// SIMATIC S7-200 SMART project (STEP 7-Micro/WIN SMART), CPU SR60

SYMBOL_TABLE Table 1
Start_0          M0.1     // Rotate the belt to fill material from the start of the belt
Start_End        M0.2     // Rotate the belt to fill material from the end of the belt
Case1            M0.3
Rotate_F         M1.3     // Rotate the shuttle trolly forward
Case3            M0.5
Case4            M0.6
Case2            M0.4
O1               M1.0
O2               M1.1
SCALED_ANALOG_INPUT VD40
Distance_in_cm   VW10     // Distance calculated by the sensor in centimeters
N1               VW20     // distance between the first sensors and the starting point of the conveyor belt
N2               VW22     // distance between the second sensors and the starting point of the conveyor belt
SENSOR_1         VW100
SENSOR_2         VW102
Rot_CW           M3.0     // Rotate the belt to fill from the start of the belt
Rot_ACW          M3.1     // Rotate the belt to fill from the end of the belt
Rotate_B         M0.7     // Rotate the shuttle trolly backword
END_SYMBOL_TABLE

SYMBOL_TABLE System Symbols
Always_On        SM0.0    // Always ON
END_SYMBOL_TABLE

ORGANIZATION_BLOCK MAIN:OB1
TITLE=Program Comments
BEGIN
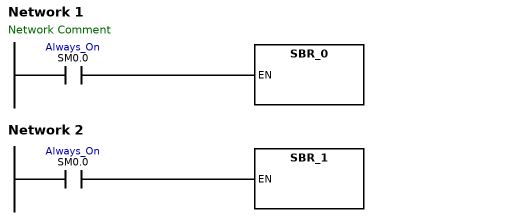
Network 1
// Network Comment
LD     Always_On:SM0.0
CALL   SBR_0:SBR0
Network 2
LD     Always_On:SM0.0
CALL   SBR_1:SBR1
END_ORGANIZATION_BLOCK

SUBROUTINE_BLOCK SBR_0:SBR0
TITLE=Subroutine Comments
BEGIN
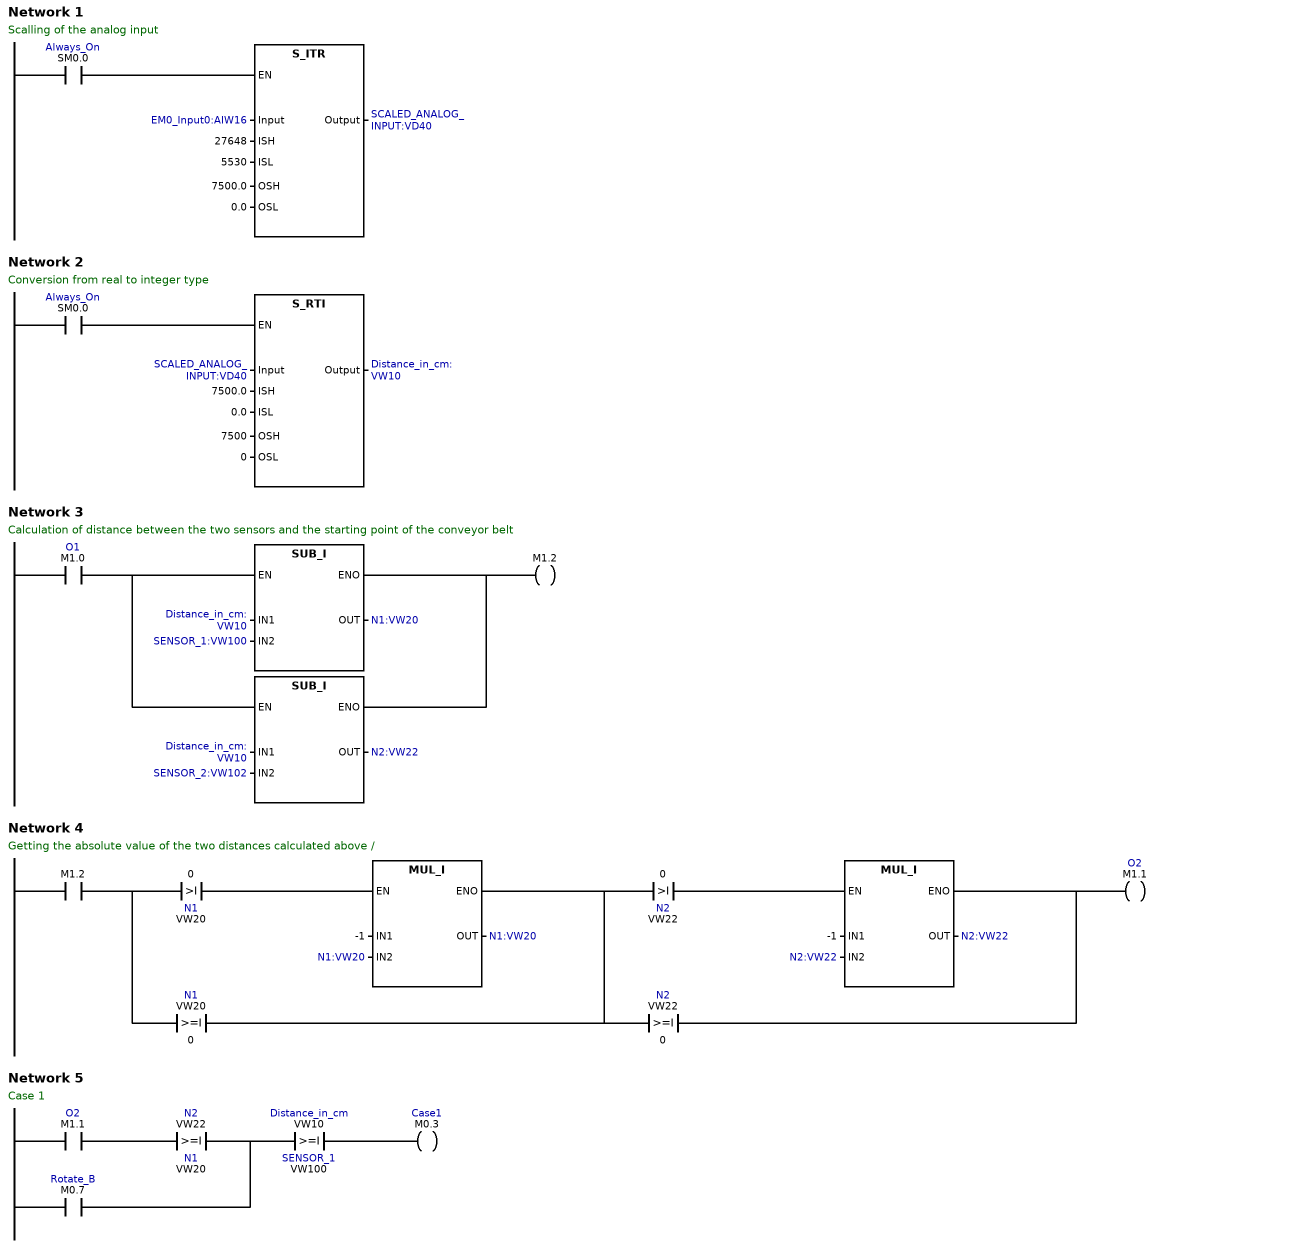
Network 1
// Scalling of the analog input
// (network saved uncompiled; LAD cells follow)
// row 0: c0 -| |- Always_On:SM0.0  c1 --  c2 [S_ITR EN:=power@row0, Input:=EM0_Input0:AIW16, ISH:=27648, ISL:=5530, OSH:=7500.0, OSL:=0.0, Output=>SCALED_ANALOG_INPUT:VD40]
// row 1: c2 [box]
// row 2: c2 [box]
Network 2
// Conversion from real to integer type
// (network saved uncompiled; LAD cells follow)
// row 0: c0 -| |- Always_On:SM0.0  c1 --  c2 [S_RTI EN:=power@row0, Input:=SCALED_ANALOG_INPUT:VD40, ISH:=7500.0, ISL:=0.0, OSH:=7500, OSL:=0, Output=>Distance_in_cm:VW10]
// row 1: c2 [box]
// row 2: c2 [box]
Network 3
// Calculation of distance between the two sensors and the starting point of the conveyor belt
// (network saved uncompiled; LAD cells follow)
// row 0: c0 -| |- O1:M1.0 v  c1 --  c2 [SUB_I EN:=power@row0, IN1:=Distance_in_cm:VW10, IN2:=SENSOR_1:VW100, ENO=>power, OUT=>N1:VW20]  c3 -- v  c4 -( ) M1.2
// row 1: c0 ^v  c2 [box]  c3 ^v
// row 2: c0 ^  c1 --  c2 [SUB_I EN:=power@row2, IN1:=Distance_in_cm:VW10, IN2:=SENSOR_2:VW102, ENO=>power, OUT=>N2:VW22]  c3 -- ^
// row 3: c2 [box]
Network 4
// Getting the absolute value of the two distances calculated above
// 
LD     M1.2
LPS
AW>    0, N1:VW20
*I     -1, N1:VW20
AENO
=      L63.7
LPP
AW>=   N1:VW20, 0
O      L63.7
LPS
AW>    0, N2:VW22
*I     -1, N2:VW22
AENO
=      L63.6
LPP
AW>=   N2:VW22, 0
O      L63.6
=      O2:M1.1
Network 5
// Case 1
// (network saved uncompiled; LAD cells follow)
// row 0: c0 -| |- O2:M1.1  c1 -|>=I|- N2:VW22, N1:VW20 v  c2 -|>=I|- Distance_in_cm:VW10, SENSOR_1:VW100  c3 -( ) Case1:M0.3
// row 1: c0 -| |- Rotate_B:M0.7  c1 -- ^
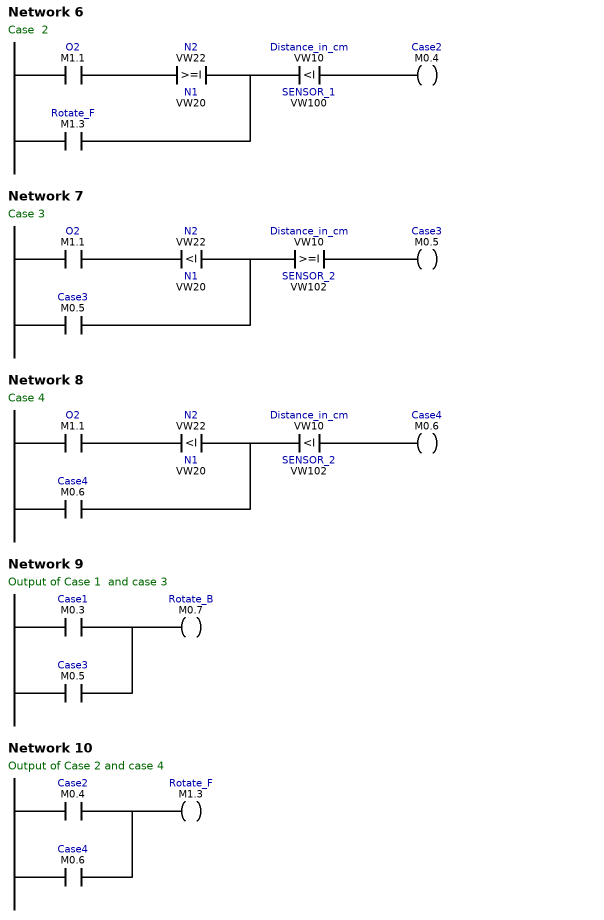
Network 6
// Case  2
// (network saved uncompiled; LAD cells follow)
// row 0: c0 -| |- O2:M1.1  c1 -|>=I|- N2:VW22, N1:VW20 v  c2 -|<I|- Distance_in_cm:VW10, SENSOR_1:VW100  c3 -( ) Case2:M0.4
// row 1: c0 -| |- Rotate_F:M1.3  c1 -- ^
Network 7
// Case 3
// (network saved uncompiled; LAD cells follow)
// row 0: c0 -| |- O2:M1.1  c1 -|<I|- N2:VW22, N1:VW20 v  c2 -|>=I|- Distance_in_cm:VW10, SENSOR_2:VW102  c3 -( ) Case3:M0.5
// row 1: c0 -| |- Case3:M0.5  c1 -- ^
Network 8
// Case 4
// (network saved uncompiled; LAD cells follow)
// row 0: c0 -| |- O2:M1.1  c1 -|<I|- N2:VW22, N1:VW20 v  c2 -|<I|- Distance_in_cm:VW10, SENSOR_2:VW102  c3 -( ) Case4:M0.6
// row 1: c0 -| |- Case4:M0.6  c1 -- ^
Network 9
// Output of Case 1  and case 3
LD     Case1:M0.3
O      Case3:M0.5
=      Rotate_B:M0.7
Network 10
// Output of Case 2 and case 4
LD     Case2:M0.4
O      Case4:M0.6
=      Rotate_F:M1.3
END_SUBROUTINE_BLOCK

SUBROUTINE_BLOCK SBR_1:SBR1
TITLE=Storage and selection of the bunker number
BEGIN
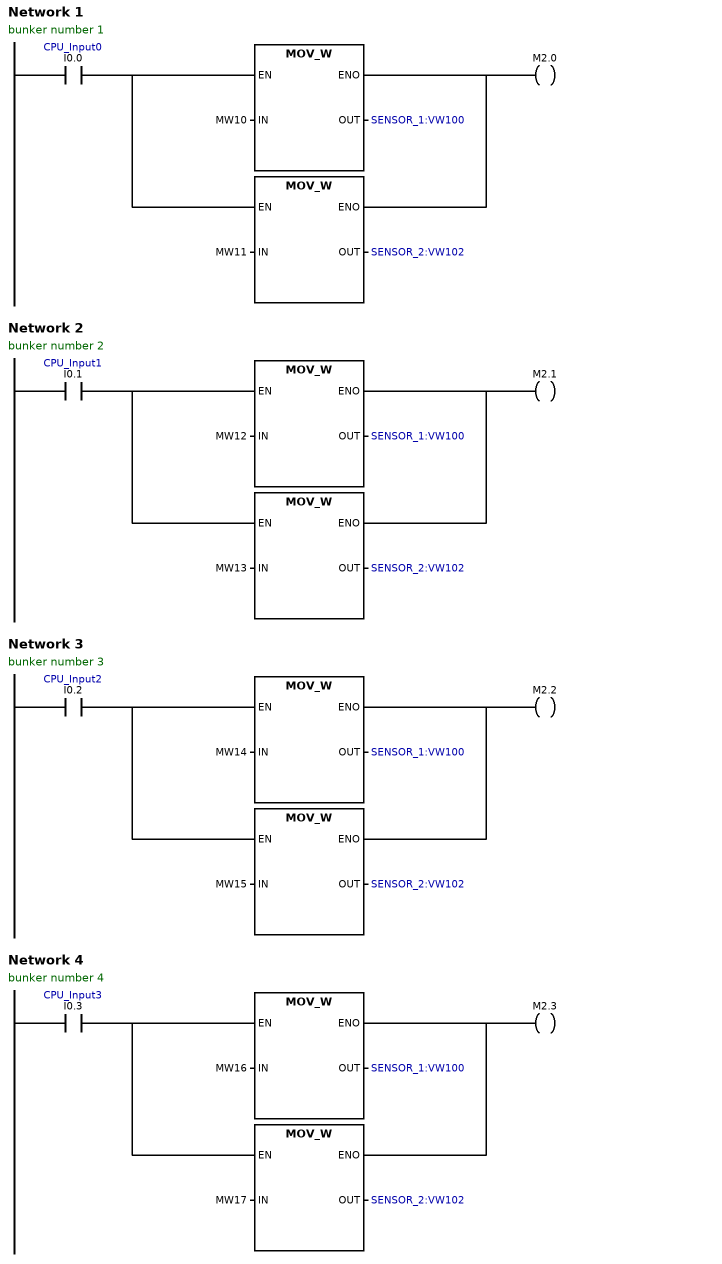
Network 1
// bunker number 1
// (network saved uncompiled; LAD cells follow)
// row 0: c0 -| |- CPU_Input0:I0.0 v  c1 --  c2 [MOV_W EN:=power@row0, IN:=MW10, ENO=>power, OUT=>SENSOR_1:VW100]  c3 -- v  c4 -( ) M2.0
// row 1: c0 ^v  c2 [box]  c3 ^v
// row 2: c0 ^  c1 --  c2 [MOV_W EN:=power@row2, IN:=MW11, ENO=>power, OUT=>SENSOR_2:VW102]  c3 -- ^
// row 3: c2 [box]
Network 2
// bunker number 2
// (network saved uncompiled; LAD cells follow)
// row 0: c0 -| |- CPU_Input1:I0.1 v  c1 --  c2 [MOV_W EN:=power@row0, IN:=MW12, ENO=>power, OUT=>SENSOR_1:VW100]  c3 -- v  c4 -( ) M2.1
// row 1: c0 ^v  c2 [box]  c3 ^v
// row 2: c0 ^  c1 --  c2 [MOV_W EN:=power@row2, IN:=MW13, ENO=>power, OUT=>SENSOR_2:VW102]  c3 -- ^
// row 3: c2 [box]
Network 3
// bunker number 3
// (network saved uncompiled; LAD cells follow)
// row 0: c0 -| |- CPU_Input2:I0.2 v  c1 --  c2 [MOV_W EN:=power@row0, IN:=MW14, ENO=>power, OUT=>SENSOR_1:VW100]  c3 -- v  c4 -( ) M2.2
// row 1: c0 ^v  c2 [box]  c3 ^v
// row 2: c0 ^  c1 --  c2 [MOV_W EN:=power@row2, IN:=MW15, ENO=>power, OUT=>SENSOR_2:VW102]  c3 -- ^
// row 3: c2 [box]
Network 4
// bunker number 4
// (network saved uncompiled; LAD cells follow)
// row 0: c0 -| |- CPU_Input3:I0.3 v  c1 --  c2 [MOV_W EN:=power@row0, IN:=MW16, ENO=>power, OUT=>SENSOR_1:VW100]  c3 -- v  c4 -( ) M2.3
// row 1: c0 ^v  c2 [box]  c3 ^v
// row 2: c0 ^  c1 --  c2 [MOV_W EN:=power@row2, IN:=MW17, ENO=>power, OUT=>SENSOR_2:VW102]  c3 -- ^
// row 3: c2 [box]
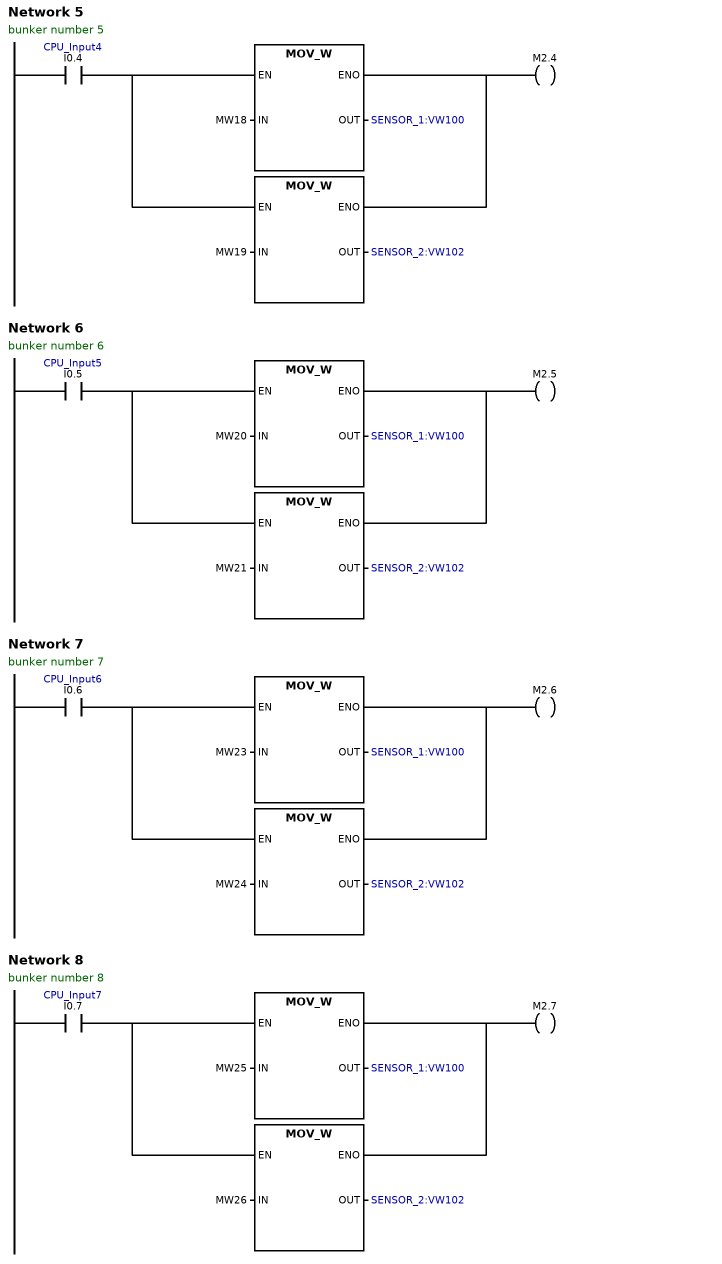
Network 5
// bunker number 5
// (network saved uncompiled; LAD cells follow)
// row 0: c0 -| |- CPU_Input4:I0.4 v  c1 --  c2 [MOV_W EN:=power@row0, IN:=MW18, ENO=>power, OUT=>SENSOR_1:VW100]  c3 -- v  c4 -( ) M2.4
// row 1: c0 ^v  c2 [box]  c3 ^v
// row 2: c0 ^  c1 --  c2 [MOV_W EN:=power@row2, IN:=MW19, ENO=>power, OUT=>SENSOR_2:VW102]  c3 -- ^
// row 3: c2 [box]
Network 6
// bunker number 6
// (network saved uncompiled; LAD cells follow)
// row 0: c0 -| |- CPU_Input5:I0.5 v  c1 --  c2 [MOV_W EN:=power@row0, IN:=MW20, ENO=>power, OUT=>SENSOR_1:VW100]  c3 -- v  c4 -( ) M2.5
// row 1: c0 ^v  c2 [box]  c3 ^v
// row 2: c0 ^  c1 --  c2 [MOV_W EN:=power@row2, IN:=MW21, ENO=>power, OUT=>SENSOR_2:VW102]  c3 -- ^
// row 3: c2 [box]
Network 7
// bunker number 7
// (network saved uncompiled; LAD cells follow)
// row 0: c0 -| |- CPU_Input6:I0.6 v  c1 --  c2 [MOV_W EN:=power@row0, IN:=MW23, ENO=>power, OUT=>SENSOR_1:VW100]  c3 -- v  c4 -( ) M2.6
// row 1: c0 ^v  c2 [box]  c3 ^v
// row 2: c0 ^  c1 --  c2 [MOV_W EN:=power@row2, IN:=MW24, ENO=>power, OUT=>SENSOR_2:VW102]  c3 -- ^
// row 3: c2 [box]
Network 8
// bunker number 8
LD     CPU_Input7:I0.7
LPS
MOVW   MW25, SENSOR_1:VW100
AENO
=      L63.7
LPP
MOVW   MW26, SENSOR_2:VW102
AENO
O      L63.7
=      M2.7
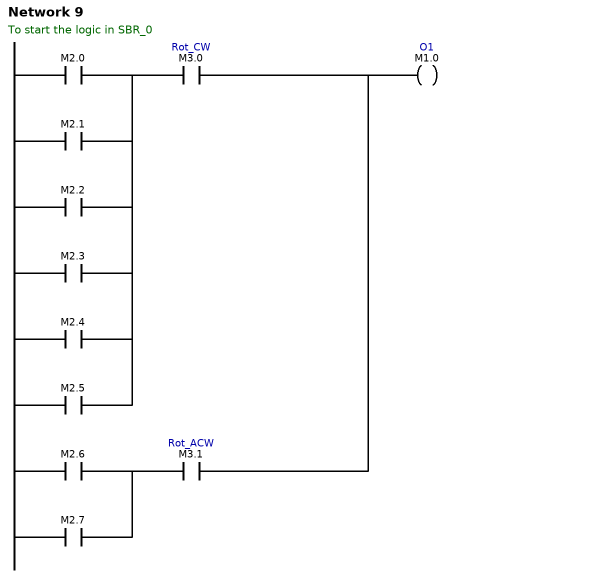
Network 9
// To start the logic in SBR_0
// (network saved uncompiled; LAD cells follow)
// row 0: c0 -| |- M2.0 v  c1 -| |- Rot_CW:M3.0  c2 -- v  c3 -( ) O1:M1.0
// row 1: c0 -| |- M2.1 ^v  c2 ^v
// row 2: c0 -| |- M2.2 ^v  c2 ^v
// row 3: c0 -| |- M2.3 ^v  c2 ^v
// row 4: c0 -| |- M2.4 ^v  c2 ^v
// row 5: c0 -| |- M2.5 ^  c2 ^v
// row 6: c0 -| |- M2.6 v  c1 -| |- Rot_ACW:M3.1  c2 -- ^
// row 7: c0 -| |- M2.7 ^
END_SUBROUTINE_BLOCK

// SBR2: protected block, not included

// SBR3: protected block, not included
